{attribute addProperty BoxType "EP3184-0002-0016"}
{attribute addProperty Id "AI_Standard_ChannelAT %I*ARRAY[0..3] OF AI_Standard_Channel_B51B79FC32440.50WcStateAT %I*WcState_98A4DF7520.250InfoDataAT %I*InfoData_BC63D37F80100"}
{attribute addProperty CRC "1907471170"}
{attribute addProperty SizeInBites "406"}
{attribute addProperty SizeInBytes "50.75"}
TYPE EP3184_360D511E :
STRUCT
	{attribute addProperty Name "AI_Standard_Channel"}
	AI_Standard_Channel : ARRAY[0..3] OF AI_Standard_Channel_B51B79FC;
	{attribute addProperty Name "WcState"}
	WcState : WcState_98A4DF75;
	{attribute addProperty Name "InfoData"}
	InfoData : InfoData_BC63D37F;
END_STRUCT
END_TYPE

(* stored: Version 1.2.0.0, ProductVersion 3.1.4024.9
   DUT EP3184_360D511E: Id {be31139b-b8eb-407a-9662-df5bb27153d2} *)
